PROGRAM MAIN
VAR
	// trigger command execution for Philips Hue samples
	bPutPhilipsHue 					: BOOL;

	fbHttpClientPhilipsHue			: FB_IotHttpClient :=(sHostName:='172.17.38.83',
									bKeepAlive:=TRUE, tConnectionTimeout:=T#10S);

	fbHttpPutPhilipsHue				: FB_TestHTTP_Put_PhilipsHue;
	
	bBlinkingMode					: BOOL;
	fbTimer							: TON:=(PT:=T#500MS);
	nColor               			: UINT;
END_VAR

// init client parameters at startup
IF NOT fbHttpClientPhilipsHue.bConfigured THEN 
	fbHttpClientPhilipsHue.nHostPort:= 80;
	fbHttpClientPhilipsHue.stTLS.bNoServerCertCheck:=TRUE;
END_IF

IF fbHttpClientPhilipsHue.bConfigured THEN
	fbHttpPutPhilipsHue(bSend:=bPutPhilipsHue, fbClient:=fbHttpClientPhilipsHue, nColor:=nColor);
END_IF

IF bBlinkingMode THEN
	fbTimer(IN:=NOT fbTimer.Q);
	IF fbTimer.Q THEN
		nColor:=nColor+5000;
		IF nColor=65000 THEN
			nColor:=0;
		END_IF
		IF bPutPhilipsHue THEN
			bPutPhilipsHue:=FALSE;
		ELSE 
			bPutPhilipsHue:=TRUE;
		END_IF
	END_IF
END_IF

fbHttpClientPhilipsHue.Execute();

END_PROGRAM

(* stored: Version 1.1.0.1, ProductVersion 3.1.4024.4
   POU MAIN: Id {e75e9aea-b793-462d-a560-528dd446e86c}, SpecialFunc None *)
